// TwinCAT 3 PLC project Sample01
// ProgramVersion: 3.1.0.8
// libraries:
//   Tc2_Standard, * (Beckhoff Automation GmbH)
//   Tc2_System, * (Beckhoff Automation GmbH)
//   Tc2_Utilities, * (Beckhoff Automation GmbH)
//   Tc3_Interfaces, * (Beckhoff Automation GmbH)
//   Tc3_MemMan, * (Beckhoff Automation GmbH)
//   Tc3_Module, * (Beckhoff Automation GmbH)
// project tree:
//   / PlcTask.TcTTO (not stored)
//   POUs/ FB_CsvLogger.TcPOU, FB_Logger.TcPOU, FB_TxtLogger.TcPOU, FB_XmlLogger.TcPOU, ILogger.TcIO, MAIN.TcPOU
// real-time tasks:
//   TASK PlcTask: cycle T#10ms, priority 20, ADS port 350

// ---- POUs/ILogger.TcIO
INTERFACE ILogger

METHOD Write : STRING
VAR_INPUT
	sMsg    : STRING;
END_VAR
END_METHOD

END_INTERFACE

// ---- POUs/FB_CsvLogger.TcPOU
{attribute 'enable_dynamic_creation'}
FUNCTION_BLOCK FB_CsvLogger IMPLEMENTS ILogger 
VAR_INPUT
END_VAR
VAR_OUTPUT
END_VAR
VAR
END_VAR

METHOD PUBLIC Write : STRING
VAR_INPUT
	sMsg      : STRING;
END_VAR
Write := CONCAT('csv-', sMsg);
// open csv file
// write the message into the csv file
// close csv file
END_METHOD

END_FUNCTION_BLOCK

// ---- POUs/FB_Logger.TcPOU
FUNCTION_BLOCK PUBLIC FB_Logger
VAR
	pTxtLogger   : POINTER TO FB_TxtLogger;
	pCsvLogger   : POINTER TO FB_CsvLogger;
	pXmlLogger   : POINTER TO FB_XmlLogger;
	ipLogger     : ILogger;
END_VAR

METHOD PUBLIC Write : STRING
VAR_INPUT
	sMsg    : STRING;
END_VAR
IF (ipLogger <> 0) THEN
	Write := ipLogger.Write(CONCAT('logger: ', sMsg));
END_IF
END_METHOD

METHOD FB_exit : BOOL
VAR_INPUT
	bInCopyCode : BOOL; // if TRUE, the exit method is called for exiting an instance that is copied afterwards (online change).
END_VAR
IF (pTxtLogger <> 0) THEN
	__DELETE(pTxtLogger);
	pTxtLogger := 0;
END_IF

IF (pCsvLogger <> 0) THEN
	__DELETE(pCsvLogger);
	pCsvLogger := 0;
END_IF

IF (pXmlLogger <> 0) THEN
	__DELETE(pXmlLogger);
	pXmlLogger := 0;
END_IF
END_METHOD

METHOD FB_init : BOOL
VAR_INPUT
    bInitRetains : BOOL; // if TRUE, the retain variables are initialized (warm start / cold start)
    bInCopyCode  : BOOL; // if TRUE, the instance afterwards gets moved into the copy code (online change)
    sFilename    : STRING;
END_VAR
VAR
	sFilenameExtension : STRING;
END_VAR
sFilenameExtension := F_ToLCase(RIGHT(sFilename, 3));
IF (sFilenameExtension = 'txt') THEN
    pTxtLogger := __NEW(FB_TxtLogger);
    ipLogger := pTxtLogger^;
ELSIF (sFilenameExtension = 'csv') THEN
    pCsvLogger := __NEW(FB_CsvLogger);
    ipLogger := pCsvLogger^;
ELSIF (sFilenameExtension = 'xml') THEN
    pXmlLogger := __NEW(FB_XmlLogger);
    ipLogger := pXmlLogger^;
ELSE
    ipLogger := 0;
END_IF
END_METHOD

END_FUNCTION_BLOCK

// ---- POUs/FB_TxtLogger.TcPOU
{attribute 'enable_dynamic_creation'}
FUNCTION_BLOCK FB_TxtLogger IMPLEMENTS ILogger
VAR_INPUT
END_VAR
VAR_OUTPUT
END_VAR
VAR
END_VAR

METHOD PUBLIC Write : STRING
VAR_INPUT
	sMsg      : STRING;
END_VAR
Write := CONCAT('txt-', sMsg);
// open txt file
// write the message into the txt file
// close txt file
END_METHOD

END_FUNCTION_BLOCK

// ---- POUs/FB_XmlLogger.TcPOU
{attribute 'enable_dynamic_creation'}
FUNCTION_BLOCK FB_XmlLogger IMPLEMENTS ILogger
VAR_INPUT
END_VAR
VAR_OUTPUT
END_VAR
VAR
END_VAR

METHOD PUBLIC Write : STRING
VAR_INPUT
	sMsg      : STRING;
END_VAR
Write := CONCAT('xml-', sMsg);
// open xml file
// write the message into the xml file
// close xml file
END_METHOD

END_FUNCTION_BLOCK

// ---- POUs/MAIN.TcPOU
PROGRAM MAIN
VAR
	fbLogger 		: FB_Logger('File.csv');
	retMsg			: STRING;
END_VAR

retMsg := fbLogger.Write('Hello');

END_PROGRAM
